{attribute 'pack_mode' := '1'}
    {attribute 'OPC.UA.DA' := '1'}
    {attribute 'OPC.UA.DA.StructuredType' := '1'}
    (*
    ST_RW_Real_HMI_IgnitionExp
    ==================================================
    Generated from Ignition UDT: RW_Real
    Total tags: 1
    Generated on: 2025-09-15 13:03:45
    *)
    TYPE ST_RW_Real_HMI_IgnitionExp :
    STRUCT
        {attribute 'OPC.UA.DA' := '1'}
        {attribute 'OPC.UA.DA.Description' := '{Description}'}
        // {Description}
        Value : REAL := 0.0;
    END_STRUCT
    END_TYPE

(* stored: Version 1.1.0.1
   DUT ST_RW_Real_HMI_IgnitionExp: Id {de0cd60b-3080-429c-ba77-75d72606e73a} *)
